FUNCTION_BLOCK L2_MachineCore (* Basic Function Block Type *)
  (* Standard: 61499-2 *)
  (* Version 0.0, 2014-11-28, EQUEROL, UJI *)
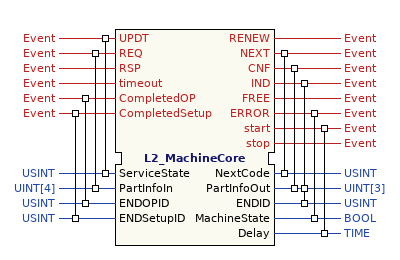
  EVENT_INPUT
    UPDT WITH ServiceState; (* Initialization Request *)
    REQ WITH PartInfoIn; (* New assignemend request *)
    RSP; (* Completed setup indication response *)
    timeout; (* timeout *)
    CompletedOP WITH ENDOPID; (* Completed operation request *)
    CompletedSetup WITH ENDSetupID; (* Current setup is done *)
  END_EVENT
  EVENT_OUTPUT
    RENEW; (* Renew Machine buffer *)
    NEXT WITH NextCode; (* Send request to execute next operation *)
    CNF WITH PartInfoOut; (* Assignement reception confirmation *)
    IND WITH PartInfoOut, ENDID; (* completed setup indication *)
    FREE; (* Indicate that the machine is free *)
    ERROR WITH MachineState; (* Indicate a change in the machine state *)
    start WITH Delay; (* Timeout start *)
    stop; (* Timeout stop *)
  END_EVENT
  VAR_INPUT
    ServiceState : USINT; (* Machine service state *)
    PartInfoIn : ARRAY [0..3] OF UINT; (* Part identifier, family and type *)
    ENDOPID : USINT := 0; (* Operation termination code *)
    ENDSetupID : USINT;
  END_VAR
  VAR_OUTPUT
    NextCode : USINT; (* Variable to indicate whixh OP must be executed next *)
    PartInfoOut : ARRAY [0..2] OF UINT; (* Part identifier, family and type *)
    ENDID : USINT; (* Setup termination code *)
    MachineState : BOOL; (* Machine state *)
    Delay : TIME; (* Timeout delay *)
  END_VAR
  VAR
    State : USINT := 1; (* Machine State *)
    CurrentPart : UINT := 0; (* Variable to contorlate the current part into the machine *)
    CurrentFamily : UINT := 0; (* Family of the current part *)
    CurrentType : UINT := 0; (* Type of the current part *)
    LostCNF : BOOL := FALSE; (* flag indicating if a trasmision error courred *)
    inError : BOOL := FALSE; (* Flag to indicate if the machine recived an error while waiting RSP *)
  END_VAR
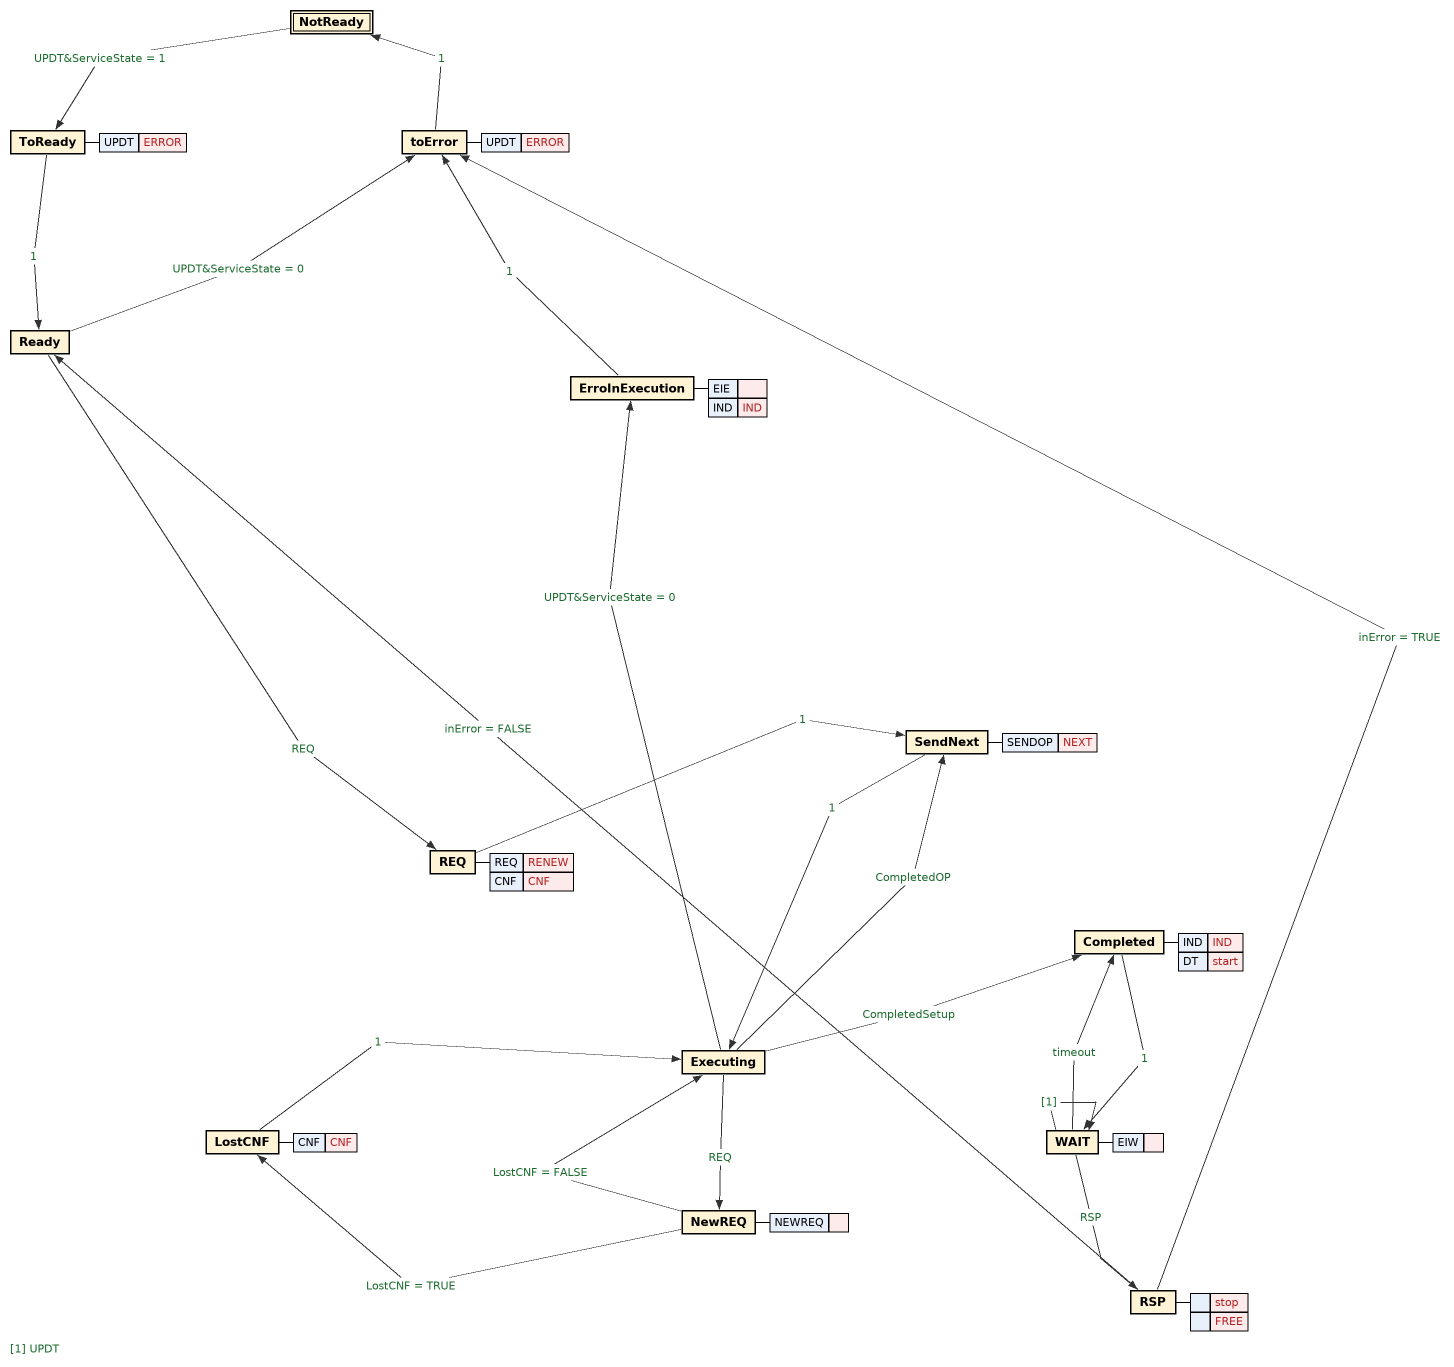
  EC_STATES
    NotReady; (* Initial State *)
    ToReady : UPDT -> ERROR;
    Ready;
    toError : UPDT -> ERROR;
    REQ : REQ -> RENEW, CNF -> CNF;
    Executing;
    Completed : IND -> IND, DT -> start;
    SendNext : SENDOP -> NEXT;
    NewREQ : NEWREQ;
    LostCNF : CNF -> CNF;
    WAIT : EIW;
    RSP : -> stop, -> FREE;
    ErroInExecution : EIE, IND -> IND;
  END_STATES
  EC_TRANSITIONS
    NotReady TO ToReady := UPDT&ServiceState = 1;
    ToReady TO Ready := 1;
    toError TO NotReady := 1;
    Ready TO toError := UPDT&ServiceState = 0;
    Ready TO REQ := REQ;
    SendNext TO Executing := 1;
    Executing TO NewREQ := REQ;
    NewREQ TO LostCNF := LostCNF = TRUE;
    LostCNF TO Executing := 1;
    NewREQ TO Executing := LostCNF = FALSE;
    Completed TO WAIT := 1;
    WAIT TO Completed := timeout;
    WAIT TO RSP := RSP;
    RSP TO Ready := inError = FALSE;
    Executing TO ErroInExecution := UPDT&ServiceState = 0;
    ErroInExecution TO toError := 1;
    WAIT TO WAIT := UPDT;
    RSP TO toError := inError = TRUE;
    Executing TO Completed := CompletedSetup;
    Executing TO SendNext := CompletedOP;
    REQ TO SendNext := 1;
  END_TRANSITIONS
  ALGORITHM REQ IN ST: (* Normally executed algorithm *)
(*A new assignation request arrived*)
(*The machine is free, confirm the assignation and modify the state*)
CurrentPart := PartInfoIn[0];
CurrentFamily := PartInfoIn[1];
CurrentType := PartInfoIn[2];
ENDOPID := 0;
  END_ALGORITHM
  ALGORITHM UPDT IN ST: (* Update machine state *)
IF ServiceState = 1 THEN
	MachineState := TRUE;
	State := 2;
ELSIF ServiceState = 0 THEN
	MachineState := FALSE;
	State := 1;
END_IF;
(*Reset inError flag every time this algo is called, It is only used in EIW*)
inError := FALSE;
  END_ALGORITHM
  ALGORITHM SENDOP IN ST: (* Send next operation algo *)
(*Post-incremented index*)
ENDOPID := NextCode;
  END_ALGORITHM
  ALGORITHM CNF IN ST: (* new algorithm *)
PartInfoOut[0] := CurrentPart;
PartInfoOut[1] := CurrentFamily;
PartInfoOut[2] := CurrentType;
  END_ALGORITHM
  ALGORITHM NEWREQ IN ST: (* new algorithm *)
(*A REQ event arrived while executing a setup*)
(*Verify if its a transmision problem or something else*)
IF CurrentPart = PartInfoIn[0] THEN
	(*Lost CNF event, retransmite it*)
	LostCNF := TRUE;
ELSE
	LostCNF := FALSE;
END_IF;
  END_ALGORITHM
  ALGORITHM DT IN ST: (* Timeout delay *)
Delay := TIME#300ms;
  END_ALGORITHM
  ALGORITHM IND IN ST: (* Completed setup indication algo *)
PartInfoOut[0] := CurrentPart;
PartInfoOut[1] := CurrentFamily;
PartInfoOut[2] := CurrentType;
ENDOPID := ENDSetupID;
  END_ALGORITHM
  ALGORITHM EIE IN ST: (* Error in execution algo *)
(*An error occurred while executing a setup*)
(*We assume that the error is not related with the setup and that it can be redone*)
ENDID := 1;
  END_ALGORITHM
  ALGORITHM EIW IN ST: (* Error in wait *)
(*An error occurred while waiting RSP*)
IF ServiceState = 0 THEN
	inError := TRUE;
END_IF;
  END_ALGORITHM
END_FUNCTION_BLOCK
